TYPE CETA_IN_u :
UNION
    bits : CETA_IN_bits_t;
    raw  : UINT;
END_UNION
END_TYPE

(* stored: Version 1.1.0.1, ProductVersion 3.1.4024.6
   DUT CETA_IN_u: Id {bb09d493-cbf2-4ce9-a0e0-be380b4acc88} *)
